{attribute 'GeneratedUsingTerminal: EL2262--0000'}
{attribute addProperty BoxType "EL2262--0000"}
{attribute addProperty Id "Cycle_CounterAT %Q*UINT2"}
{attribute addProperty CRC "740505604"}
{attribute addProperty Size "2"}
TYPE Cycle_Counter_2C233804 EXTENDS OutputBase_10CEE7DE :
STRUCT
	{attribute addProperty Name "Cycle_Counter"}
	Cycle_Counter AT %Q* : UINT;
END_STRUCT
END_TYPE

(* stored: Version 1.2.0.0, ProductVersion 3.1.4024.9
   DUT Cycle_Counter_2C233804: Id {69cffed0-a03e-4fe4-a692-04edebd3c721} *)
